TYPE ST_OffScreenTest :
STRUCT	

	//enter Single Joint test mode
	m_enterOffScreenTestMode:ARRAY[1..g_sArmNum] OF BOOL;
	m_singleJntFlag,m_return2OriginFlag,m_move2StartFlag:BOOL;
	m_kineCaliJntIdx:INT:=0;
	
	m_caliPointStartFlag:ARRAY[1..9] OF BOOL := [9(FALSE)];
	m_caliPointEndFlag:ARRAY[1..9] OF BOOL := [9(TRUE)];
	
	m_dataRecordFlag:ARRAY[1..g_sArmNum] OF BOOL:=[4(FALSE)];
	m_dataRecordCount:ARRAY[1..g_sArmNum] OF INT:=[4(0)];
	m_dataSingleCount:INT:=0;
	m_dataShowCount:STRING:='0';
	m_dataRecordText:STRING := 'No record';

	
END_STRUCT
END_TYPE

(* stored: Version 1.1.0.1, ProductVersion 3.1.4024.11
   DUT ST_OffScreenTest: Id {a8c6a6f1-dce6-473b-ab0c-062c11b2196d} *)
